// TIA Portal V17 export
// export: Created 2023-04-06T14:59:51.4519566Z, ExportSetting None, DisplayName Totally Integrated Automation Portal, DisplayVersion V17 Update 4, DisplayName TIA Portal Openness, DisplayVersion V17 Update 4, DisplayName TIA Portal Version Control Interface, DisplayVersion V17, DisplayName STEP 7 Professional, DisplayVersion V17 Update 4, DisplayName STEP 7 Safety, DisplayVersion V17, DisplayName WinCC Advanced / Unified PC, DisplayVersion V17 Update 4
DATA_BLOCK "SETTINGS"   // DB25
{ S7_Optimized_Access := 'FALSE' }
// stored: AutoNumber false
   VAR RETAIN
      PT_1 : Struct   // MAIN RING SYSTEM PRESSURE
         RANGE_L : Real := 0.0;
         RANGE_H : Real := 100.0;
         SP_LL : Real := -1000.0;
         SP_L : Real := -1000.0;
         SP_H : Real := 1000.0;
         SP_HH : Real := 1000.0;
      END_STRUCT;
      FT_1 : Struct   // MAIN RING FLOW
         RANGE_L : Real := 0.0;
         RANGE_H : Real := 200.0;
         SP_LL : Real := -1000.0;
         SP_L : Real := -1000.0;
         SP_H : Real := 1000.0;
         SP_HH : Real := 1000.0;
      END_STRUCT;
      FT_2 : Struct   // INGERSOL COMPRESSOR OUTLET FLOW
         RANGE_L : Real := 0.0;
         RANGE_H : Real := 300.0;
         SP_LL : Real := -1000.0;
         SP_L : Real := -1000.0;
         SP_H : Real := 1000.0;
         SP_HH : Real := 1000.0;
      END_STRUCT;
      FT_3 : Struct   // HANWA COMPRESSOR 1 OUTLET FLOW
         RANGE_L : Real := 0.0;
         RANGE_H : Real := 400.0;
         SP_LL : Real := -1000.0;
         SP_L : Real := -1000.0;
         SP_H : Real := 1000.0;
         SP_HH : Real := 1000.0;
      END_STRUCT;
      FT_4 : Struct   // HANWA COMPRESSOR 2 OUTLET FLOW
         RANGE_L : Real := 0.0;
         RANGE_H : Real := 500.0;
         SP_LL : Real := -1000.0;
         SP_L : Real := -1000.0;
         SP_H : Real := 1000.0;
         SP_HH : Real := 1000.0;
      END_STRUCT;
      FT_5 : Struct   // HIGH PRESSURE RING FLOW
         RANGE_L : Real := 0.0;
         RANGE_H : Real := 600.0;
         SP_LL : Real := -1000.0;
         SP_L : Real := -1000.0;
         SP_H : Real := 1000.0;
         SP_HH : Real := 1000.0;
      END_STRUCT;
      FT_6 : Struct   // HIGH PRESSURE RING FLOW
         RANGE_L : Real := 0.0;
         RANGE_H : Real := 700.0;
         SP_LL : Real := -1000.0;
         SP_L : Real := -1000.0;
         SP_H : Real := 1000.0;
         SP_HH : Real := 1000.0;
      END_STRUCT;
   END_VAR
BEGIN
END_DATA_BLOCK
